{attribute 'qualified_only' := ''}
{attribute 'strict' := ''}
{attribute 'to_string' := ''}
TYPE cLaneSel :
(
	None := 0,
	Green := 1,
	Red := 2,
	Blue := 3
);
END_TYPE

(* stored: Version 1.1.0.1, ProductVersion 3.1.4024.6
   DUT cLaneSel: Id {8885da5a-af8c-4e9e-9283-3f0b431f0250} *)
